(* PLC project Untitled1, Eclipse Foundation CIF to Structured Text 0.0 *)
(* stored: creationDateTime 1970-01-01T00:00:00Z *)

PROGRAM MAIN
  VAR
    p_x : DINT;
    p_t : REAL;
    preset_p_t : TIME;
    firstRun : BOOL := TRUE;
    loopsKilled : INT;
  END_VAR
  VAR_TEMP
    loopCount : DINT;
    curValue : REAL;
    current_p_t : REAL;
    edge_p_1 : DINT;
    eventEnabled : BOOL;
    isProgress : BOOL;
    timeOut : BOOL;
  END_VAR

            (* Header text file for:
 *  -> (-*-) CIF PLC code generator.
 *)

(* --- Initialize state or update continuous variables. -------------------- *)
IF firstRun THEN
    firstRun := FALSE;
    loopsKilled := 0;

    (* Initialize the state variables. *)
    p_x := 5;
    p_t := 0.0;
    (* Reset timer of "p_t". *)
    preset_p_t := p_t;
    ton_p_t(IN := FALSE, PT := preset_p_t);
    ton_p_t(IN := TRUE, PT := preset_p_t);
ELSE
    (* Update remaining time of "p_t". *)
    ton_p_t(IN := TRUE, PT := preset_p_t, Q => timeOut, ET => curValue);
    p_t := SEL(timeOut, preset_p_t - curValue, 0.0);
END_IF;

(* --- Process uncontrollable events. -------------------------------------- *)
isProgress := TRUE;
(* Perform events until none can be done anymore. *)
(* Track the number of iterations and abort if there are too many. *)
loopCount := 0;
WHILE isProgress AND loopCount < 101 DO
    loopCount := loopCount + 1;
    isProgress := FALSE;

    (*************************************************************
     * Try to perform event "e".
     *
     * - Automaton "p" must always synchronize.
     *************************************************************)
    eventEnabled := TRUE;
    (*******************************
     * Check each synchronizing automaton for having an edge with a true guard.
     *******************************)
    (***********
     * Testing edge of automaton "p" to synchronize for event "e".
     * This automaton must have an edge with a true guard to allow the event.
     *
     * Edge being tested:
     * - Location:
     *   - 1st edge in the location
     ***********)
    IF p_t <= 1.0 AND p_x = 5 THEN
        edge_p_1 := 1;
    ELSE
        (* The automaton has no edge with a true guard. Skip to the next event. *)
        eventEnabled := FALSE;
    END_IF;
    (* All checks have been done. If variable "eventEnabled" still holds, event "e" can occur. *)
    IF eventEnabled THEN
        isProgress := TRUE;
        (* Make temporary copies of assigned variables to preserve the old values while assigning new values. *)
        current_p_t := p_t;
        (*******************************
         * Perform the assignments of each synchronizing automaton.
         *******************************)
        (* Perform assignments of automaton "p". *)
        IF edge_p_1 = 1 THEN
            (* Perform assignments of the 1st edge of automaton "p". *)
            p_t := 7.0;
            (* Reset timer of "p_t". *)
            preset_p_t := p_t;
            ton_p_t(IN := FALSE, PT := preset_p_t);
            ton_p_t(IN := TRUE, PT := preset_p_t);
        END_IF;
    END_IF;
END_WHILE;
(* Register the first 9999 aborted loops. *)
IF loopCount >= 101 THEN
    loopsKilled := MIN(loopsKilled + 1, 9999);
END_IF;
          
END_PROGRAM

CONFIGURATION Untitled1
  RESOURCE Untitled1 ON PLC
    VAR_GLOBAL  (* TIMERS *)
      ton_p_t : TON;
    END_VAR
    TASK PlcTask(INTERVAL := T#0ms, PRIORITY := 20);
    PROGRAM MAIN WITH PlcTask : MAIN;
  END_RESOURCE
END_CONFIGURATION
